(*
Allows registration of FB implementing `I_Component`. The framework will automatically add this function block to the entity's scope.
*)
FUNCTION_BLOCK FINAL Component IMPLEMENTS I_Component
VAR
	_iComponent: I_RawComponent;
	_iEntity: I_Entity;
	_iNext: I_Component;
	_iPrev: I_Component;			
END_VAR

PROPERTY _AsiComponent : I_Component
GET
_AsIComponent := THIS^;
END_GET
END_PROPERTY

PROPERTY _Entity : I_Entity
GET
_Entity := _iEntity;
END_GET
SET
_iEntity := _Entity;
END_SET
END_PROPERTY

PROPERTY _Next : I_ComponentNode
GET
_Next := _iNext;
END_GET
SET
_iNext := _Next._AsiComponent;
END_SET
END_PROPERTY

PROPERTY _Prev : I_ComponentNode
GET
_Prev := _iPrev;
END_GET
SET
_iPrev := _Prev._AsiComponent;
END_SET
END_PROPERTY

(*
Returns parent Entity.
*)
PROPERTY Entity : I_Entity
GET
Entity := _iEntity;
END_GET
END_PROPERTY

//FB_Init is always available implicitly and it is used primarily for initialization.
//The return value is not evaluated. For a specific influence, you can also declare the
//methods explicitly and provide additional code there with the standard initialization
//code. You can evaluate the return value.
{attribute 'hide'}
METHOD FB_init: BOOL
VAR_INPUT
    bInitRetains: BOOL; // TRUE: the retain variables are initialized (reset warm / reset cold)
    bInCopyCode: BOOL;  // TRUE: the instance will be copied to the copy code afterward (online change)
	
	iComponent		: I_RawComponent;
END_VAR
VAR
	_nResult		: Result;
END_VAR
_iComponent := iComponent;

IF _Ec.iUnderConstruction = 0 THEN
	DebugMsg(THIS^, 'Declared outside Entity scope!');
	RETURN;
END_IF
			
IF IsErr(_RegisterComponent(THIS^), nOut => _nResult) THEN
	DebugMsg(THIS^, Tc2_Standard.CONCAT('Failed with code: ', ResultToStr(_nResult)));
END_IF
END_METHOD

(*
Returns raw I_Component pointer.
*)
PROPERTY Raw : I_RawComponent
GET
Raw := _iComponent;
END_GET
END_PROPERTY

END_FUNCTION_BLOCK

(* stored: Version 1.1.0.1
   POU Component: Id {fa960ebd-c1a5-43b6-93f9-37986edc8a8e}, SpecialFunc None
   Folder _: Id {2f64ab46-31e6-48ed-9d95-c4291bcfd948}
   Property _AsiComponent: Id {47b9770d-a779-430d-8c42-5bfef0941f79}
   Get Get: Id {4a4979e6-2905-4c2b-a12f-d659a7c19d62}
   Property _Entity: Id {04992c4b-8576-490a-bc5a-4ea7e42d0690}
   Get Get: Id {4099a2bf-0181-4f7e-83da-372c0e5753e4}
   Set Set: Id {5c120199-3d0f-4c55-aed9-23d3550af9a3}
   Property _Next: Id {b697f57c-1907-4eab-afeb-f88c92893472}
   Get Get: Id {fbe2d6bf-25b1-49dd-b699-6801a0cd8f57}
   Set Set: Id {7f04b85c-87a9-43e1-ad09-8aa8b8f0995e}
   Property _Prev: Id {49dba3a3-71ab-4665-bf1c-df44eb849e53}
   Get Get: Id {5188ba92-1868-49bb-ac7c-116358111ebe}
   Set Set: Id {312bfdfd-5d0b-428d-a350-b64bcdfbc76b}
   Property Entity: Id {03f954b7-96dd-486d-bc2c-304b7fa3fabf}
   Get Get: Id {d240c28c-91c6-4daa-8272-834d768826b4}
   Method FB_init: Id {6b3be823-b707-4752-9ff4-9bf296045f36}
   Property Raw: Id {f0629eb7-2548-4aad-92a4-4ae12d6f0db5}
   Get Get: Id {ce00bc59-cc2a-41f7-9580-773a33558064} *)
